{attribute 'linkalways'} 
{attribute 'no_explicit_call' := 'This FB is a CLASS and must be accessed using methods or properties'}
{attribute 'enable_dynamic_creation'}
FUNCTION_BLOCK PUBLIC ResetCommand EXTENDS AxisCommand

METHOD FB_init : BOOL
VAR_INPUT
	bInitRetains : BOOL; // if TRUE, the retain variables are initialized (warm start / cold start)
	bInCopyCode : BOOL;  // if TRUE, the instance afterwards gets moved into the copy code (online change)
	axis : I_Axis;
END_VAR
_axis := axis;
END_METHOD

METHOD PROTECTED OnExecuting
VAR_INPUT
	stateControl : I_AsyncCommandStateControl;
END_VAR
VAR_INST
	_fb : MC_Reset;
END_VAR
_fb(
	Axis := _axis._InternalAxisRef,
	Execute := TRUE
);

IF _fb.Busy THEN
	RETURN;
END_IF

_fb(Axis := _axis._InternalAxisRef, Execute := FALSE);

IF _fb.Error THEN
	stateControl.Error(_fb.ErrorID);
	RETURN;
END_IF

stateControl.Next();
END_METHOD

END_FUNCTION_BLOCK

(* stored: Version 1.1.0.1, ProductVersion 3.1.4024.12
   POU ResetCommand: Id {fbdd2803-8795-42d1-8ee7-9a961a7284c0}, SpecialFunc None
   Folder Constructor: Id {ee8f912a-5352-4190-88f7-9f07ef07cd8a}
   Method FB_init: Id {8faec425-f017-4414-8fa5-d98a0fc8bdd1}
   Method OnExecuting: Id {9282fbef-f337-0c94-0ea6-eda9ca8d322c} *)
